{attribute 'GeneratedUsingTerminal: EM7004-0000-0017'}
{attribute addProperty BoxType "EM7004-0000-0017"}
{attribute addProperty Id "Output_0BOOL1Output_1BOOL1Output_2BOOL1Output_3BOOL1Output_4BOOL1Output_5BOOL1Output_6BOOL1Output_7BOOL1Output_8BOOL1Output_9BOOL1Output_10BOOL1Output_11BOOL1Output_12BOOL1Output_13BOOL1Output_14BOOL1Output_15BOOL1"}
{attribute addProperty CRC "4294934650"}
{attribute addProperty Size "16"}
TYPE Output_FFFF807A :
STRUCT
	{attribute addProperty Name "Output_0"}
	Output_0 : BOOL;
	{attribute addProperty Name "Output_1"}
	Output_1 : BOOL;
	{attribute addProperty Name "Output_2"}
	Output_2 : BOOL;
	{attribute addProperty Name "Output_3"}
	Output_3 : BOOL;
	{attribute addProperty Name "Output_4"}
	Output_4 : BOOL;
	{attribute addProperty Name "Output_5"}
	Output_5 : BOOL;
	{attribute addProperty Name "Output_6"}
	Output_6 : BOOL;
	{attribute addProperty Name "Output_7"}
	Output_7 : BOOL;
	{attribute addProperty Name "Output_8"}
	Output_8 : BOOL;
	{attribute addProperty Name "Output_9"}
	Output_9 : BOOL;
	{attribute addProperty Name "Output_10"}
	Output_10 : BOOL;
	{attribute addProperty Name "Output_11"}
	Output_11 : BOOL;
	{attribute addProperty Name "Output_12"}
	Output_12 : BOOL;
	{attribute addProperty Name "Output_13"}
	Output_13 : BOOL;
	{attribute addProperty Name "Output_14"}
	Output_14 : BOOL;
	{attribute addProperty Name "Output_15"}
	Output_15 : BOOL;
END_STRUCT
END_TYPE

(* stored: Version 1.2.0.0, ProductVersion 3.1.4024.9
   DUT Output_FFFF807A: Id {cd7b6894-5c02-4bc0-ab95-2176cba51bcf} *)
